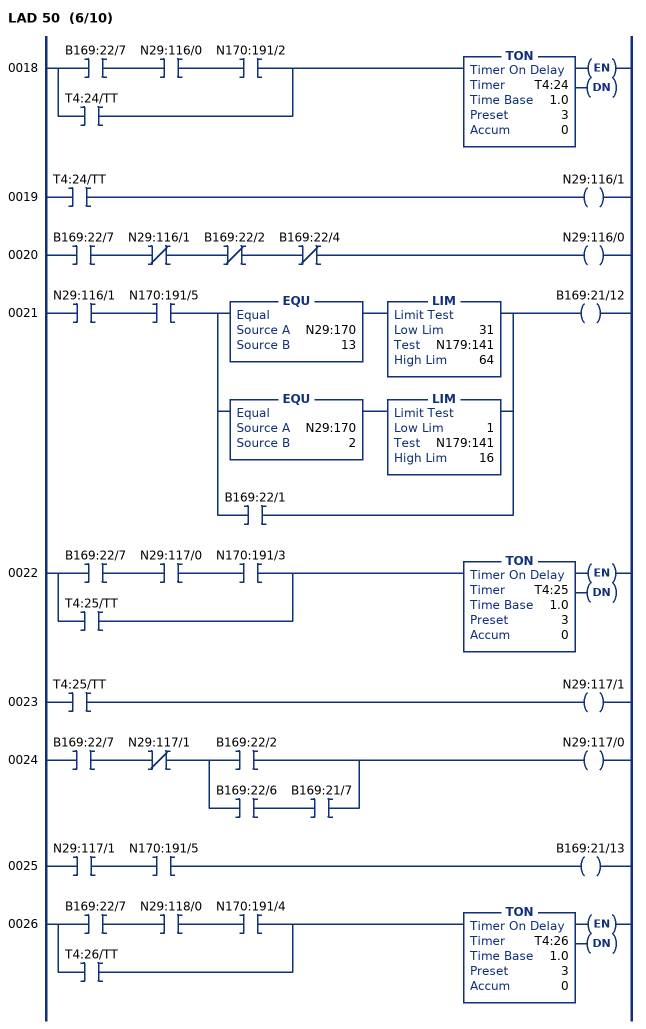
% Rung: 18 %
SOR BST XIC B169:22/7 XIC N29:116/0 XIC N170:191/2 NXB XIC T4:24/TT BND TON T4:24 1.0 3 0 EOR
% Rung: 19 %
SOR XIC T4:24/TT OTE N29:116/1 EOR
% Rung: 20 %
SOR XIC B169:22/7 XIO N29:116/1 XIO B169:22/2 XIO B169:22/4 OTE N29:116/0 EOR
% Rung: 21 %
SOR XIC N29:116/1 XIC N170:191/5 BST EQU N29:170 13 LIM 31 N179:141 64 NXB EQU N29:170 2 LIM 1 N179:141 16 NXB XIC B169:22/1 BND OTE B169:21/12 EOR
% Rung: 22 %
SOR BST XIC B169:22/7 XIC N29:117/0 XIC N170:191/3 NXB XIC T4:25/TT BND TON T4:25 1.0 3 0 EOR
% Rung: 23 %
SOR XIC T4:25/TT OTE N29:117/1 EOR
% Rung: 24 %
SOR XIC B169:22/7 XIO N29:117/1 BST XIC B169:22/2 NXB XIC B169:22/6 XIC B169:21/7 BND OTE N29:117/0 EOR
% Rung: 25 %
SOR XIC N29:117/1 XIC N170:191/5 OTE B169:21/13 EOR
% Rung: 26 %
SOR BST XIC B169:22/7 XIC N29:118/0 XIC N170:191/4 NXB XIC T4:26/TT BND TON T4:26 1.0 3 0 EOR

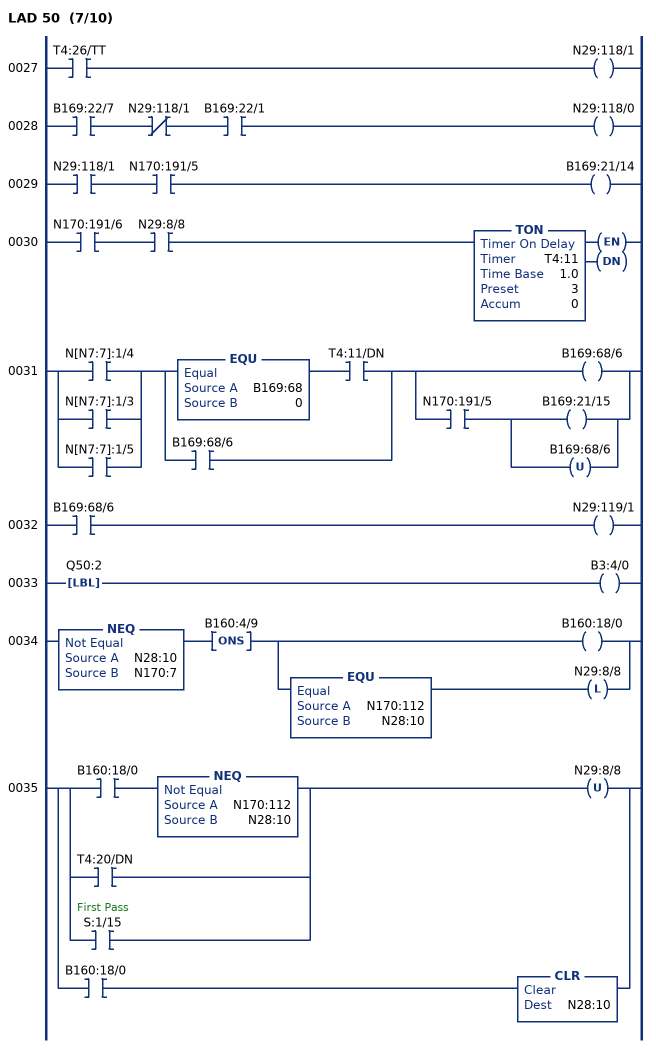
% Rung: 27 %
SOR XIC T4:26/TT OTE N29:118/1 EOR
% Rung: 28 %
SOR XIC B169:22/7 XIO N29:118/1 XIC B169:22/1 OTE N29:118/0 EOR
% Rung: 29 %
SOR XIC N29:118/1 XIC N170:191/5 OTE B169:21/14 EOR
% Rung: 30 %
SOR XIC N170:191/6 XIC N29:8/8 TON T4:11 1.0 3 0 EOR
% Rung: 31 %
SOR BST XIC N[N7:7]:1/4 NXB XIC N[N7:7]:1/3 NXB XIC N[N7:7]:1/5 BND BST EQU B169:68 0 XIC T4:11/DN NXB XIC B169:68/6 BND BST OTE B169:68/6 NXB XIC N170:191/5 BST OTE B169:21/15 NXB OTU B169:68/6 BND BND EOR
% Rung: 32 %
SOR XIC B169:68/6 OTE N29:119/1 EOR
% Rung: 33 %
SOR LBL Q50:2 OTE B3:4/0 EOR
% Rung: 34 %
SOR NEQ N28:10 N170:7 OSR B160:4/9 BST OTE B160:18/0 NXB EQU N170:112 N28:10 OTL N29:8/8 BND EOR
% Rung: 35 %
SOR BST BST XIC B160:18/0 NEQ N170:112 N28:10 NXB XIC T4:20/DN NXB XIC S:1/15 BND OTU N29:8/8 NXB XIC B160:18/0 CLR N28:10 BND EOR
%   S:1/15  "First Pass" %

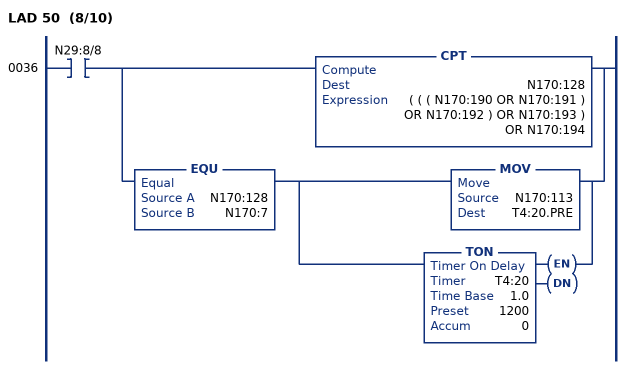
% Rung: 36 %
SOR XIC N29:8/8 BST CPT N170:128 " ( ( ( N170:190 OR N170:191 ) OR N170:192 ) OR N170:193 ) OR N170:194 " NXB EQU N170:128 N170:7 BST MOV N170:113 T4:20.PRE NXB TON T4:20 1.0 1200 0 BND BND EOR

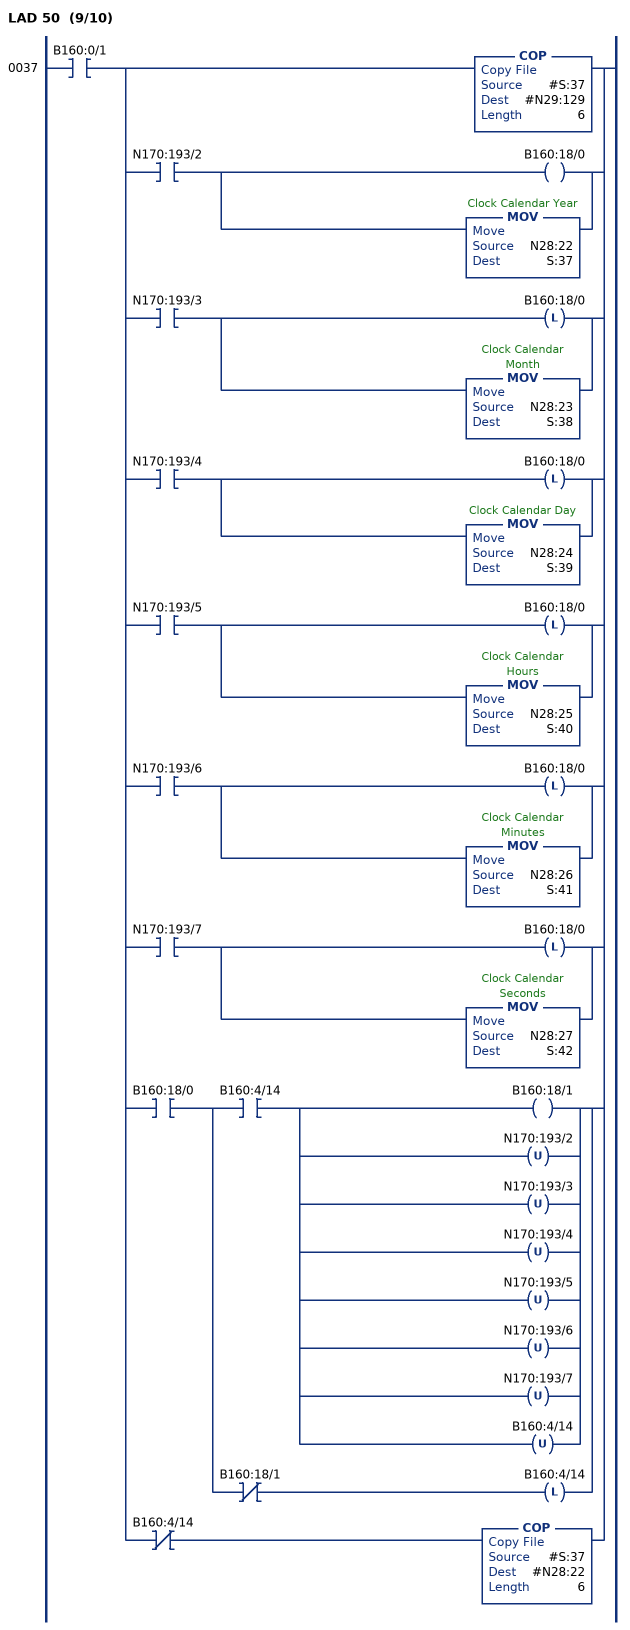
% Rung: 37 %
SOR XIC B160:0/1 BST COP #S:37 #N29:129 6 NXB XIC N170:193/2 BST OTE B160:18/0 NXB MOV N28:22 S:37 BND NXB XIC N170:193/3 BST OTL B160:18/0 NXB MOV N28:23 S:38 BND NXB XIC N170:193/4 BST OTL B160:18/0 NXB MOV N28:24 S:39 BND NXB XIC N170:193/5 BST OTL B160:18/0 NXB MOV N28:25 S:40 BND NXB XIC N170:193/6 BST OTL B160:18/0 NXB MOV N28:26 S:41 BND NXB XIC N170:193/7 BST OTL B160:18/0 NXB MOV N28:27 S:42 BND NXB XIC B160:18/0 BST XIC B160:4/14 BST OTE B160:18/1 NXB OTU N170:193/2 NXB OTU N170:193/3 NXB OTU N170:193/4 NXB OTU N170:193/5 NXB OTU N170:193/6 NXB OTU N170:193/7 NXB OTU B160:4/14 BND NXB XIO B160:18/1 OTL B160:4/14 BND NXB XIO B160:4/14 COP #S:37 #N28:22 6 BND EOR
%   S:37  "Clock Calendar Year" %
%   S:38  "Clock Calendar Month" %
%   S:39  "Clock Calendar Day" %
%   S:40  "Clock Calendar Hours" %
%   S:41  "Clock Calendar Minutes" %
%   S:42  "Clock Calendar Seconds" %

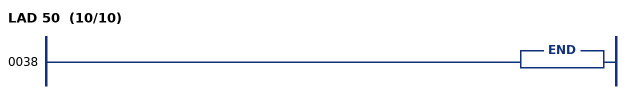
% Rung: 38 %
SOR END EOR

LADDER 51
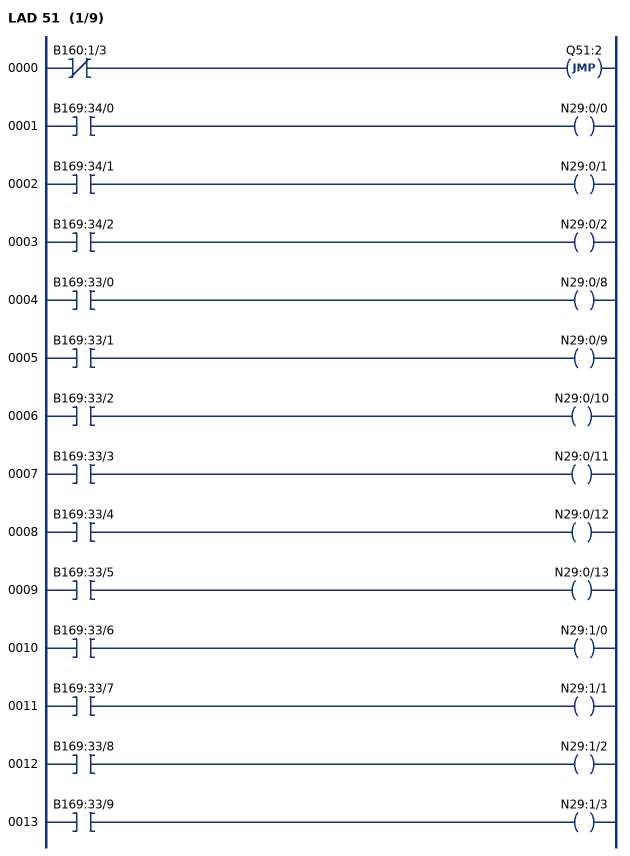
% Rung: 0 %
SOR XIO B160:1/3 JMP Q51:2 EOR
% Rung: 1 %
SOR XIC B169:34/0 OTE N29:0/0 EOR
% Rung: 2 %
SOR XIC B169:34/1 OTE N29:0/1 EOR
% Rung: 3 %
SOR XIC B169:34/2 OTE N29:0/2 EOR
% Rung: 4 %
SOR XIC B169:33/0 OTE N29:0/8 EOR
% Rung: 5 %
SOR XIC B169:33/1 OTE N29:0/9 EOR
% Rung: 6 %
SOR XIC B169:33/2 OTE N29:0/10 EOR
% Rung: 7 %
SOR XIC B169:33/3 OTE N29:0/11 EOR
% Rung: 8 %
SOR XIC B169:33/4 OTE N29:0/12 EOR
% Rung: 9 %
SOR XIC B169:33/5 OTE N29:0/13 EOR
% Rung: 10 %
SOR XIC B169:33/6 OTE N29:1/0 EOR
% Rung: 11 %
SOR XIC B169:33/7 OTE N29:1/1 EOR
% Rung: 12 %
SOR XIC B169:33/8 OTE N29:1/2 EOR
% Rung: 13 %
SOR XIC B169:33/9 OTE N29:1/3 EOR

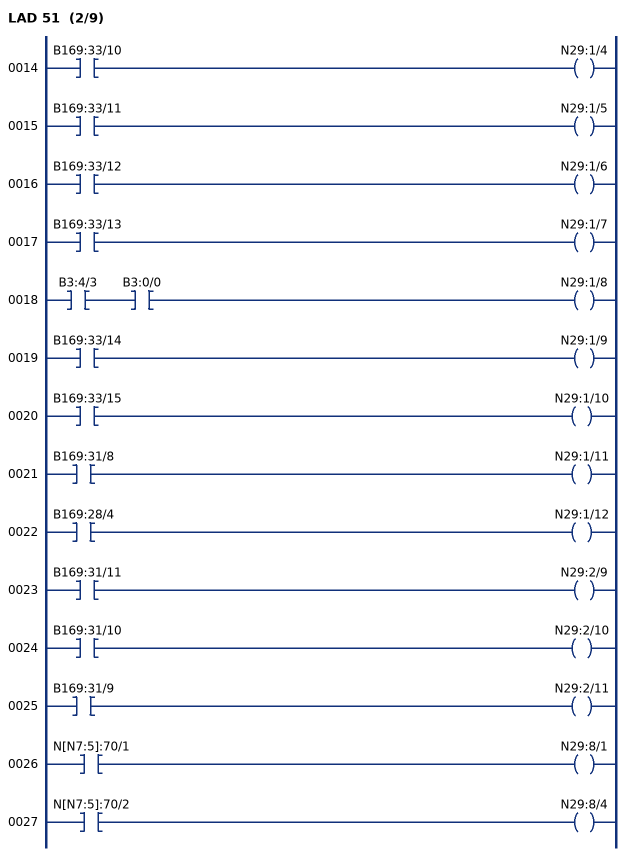
% Rung: 14 %
SOR XIC B169:33/10 OTE N29:1/4 EOR
% Rung: 15 %
SOR XIC B169:33/11 OTE N29:1/5 EOR
% Rung: 16 %
SOR XIC B169:33/12 OTE N29:1/6 EOR
% Rung: 17 %
SOR XIC B169:33/13 OTE N29:1/7 EOR
% Rung: 18 %
SOR XIC B3:4/3 XIC B3:0/0 OTE N29:1/8 EOR
% Rung: 19 %
SOR XIC B169:33/14 OTE N29:1/9 EOR
% Rung: 20 %
SOR XIC B169:33/15 OTE N29:1/10 EOR
% Rung: 21 %
SOR XIC B169:31/8 OTE N29:1/11 EOR
% Rung: 22 %
SOR XIC B169:28/4 OTE N29:1/12 EOR
% Rung: 23 %
SOR XIC B169:31/11 OTE N29:2/9 EOR
% Rung: 24 %
SOR XIC B169:31/10 OTE N29:2/10 EOR
% Rung: 25 %
SOR XIC B169:31/9 OTE N29:2/11 EOR
% Rung: 26 %
SOR XIC N[N7:5]:70/1 OTE N29:8/1 EOR
% Rung: 27 %
SOR XIC N[N7:5]:70/2 OTE N29:8/4 EOR

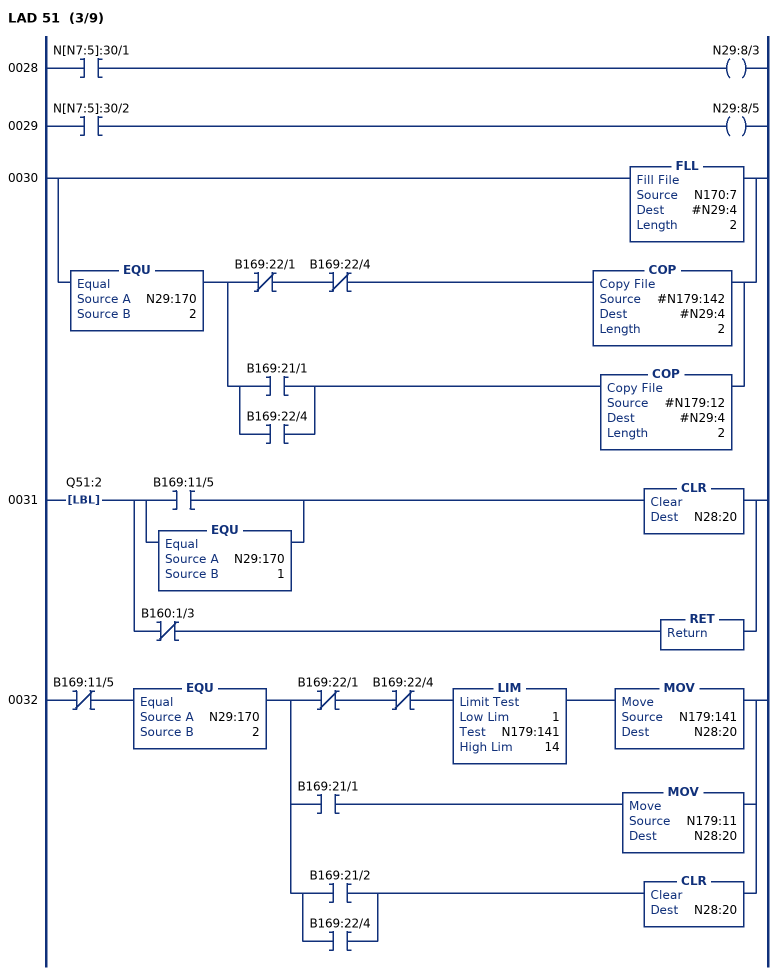
% Rung: 28 %
SOR XIC N[N7:5]:30/1 OTE N29:8/3 EOR
% Rung: 29 %
SOR XIC N[N7:5]:30/2 OTE N29:8/5 EOR
% Rung: 30 %
SOR BST FLL N170:7 #N29:4 2 NXB EQU N29:170 2 BST XIO B169:22/1 XIO B169:22/4 COP #N179:142 #N29:4 2 NXB BST XIC B169:21/1 NXB XIC B169:22/4 BND COP #N179:12 #N29:4 2 BND BND EOR
% Rung: 31 %
SOR LBL Q51:2 BST BST XIC B169:11/5 NXB EQU N29:170 1 BND CLR N28:20 NXB XIO B160:1/3 RET BND EOR
% Rung: 32 %
SOR XIO B169:11/5 EQU N29:170 2 BST XIO B169:22/1 XIO B169:22/4 LIM 1 N179:141 14 MOV N179:141 N28:20 NXB XIC B169:21/1 MOV N179:11 N28:20 NXB BST XIC B169:21/2 NXB XIC B169:22/4 BND CLR N28:20 BND EOR

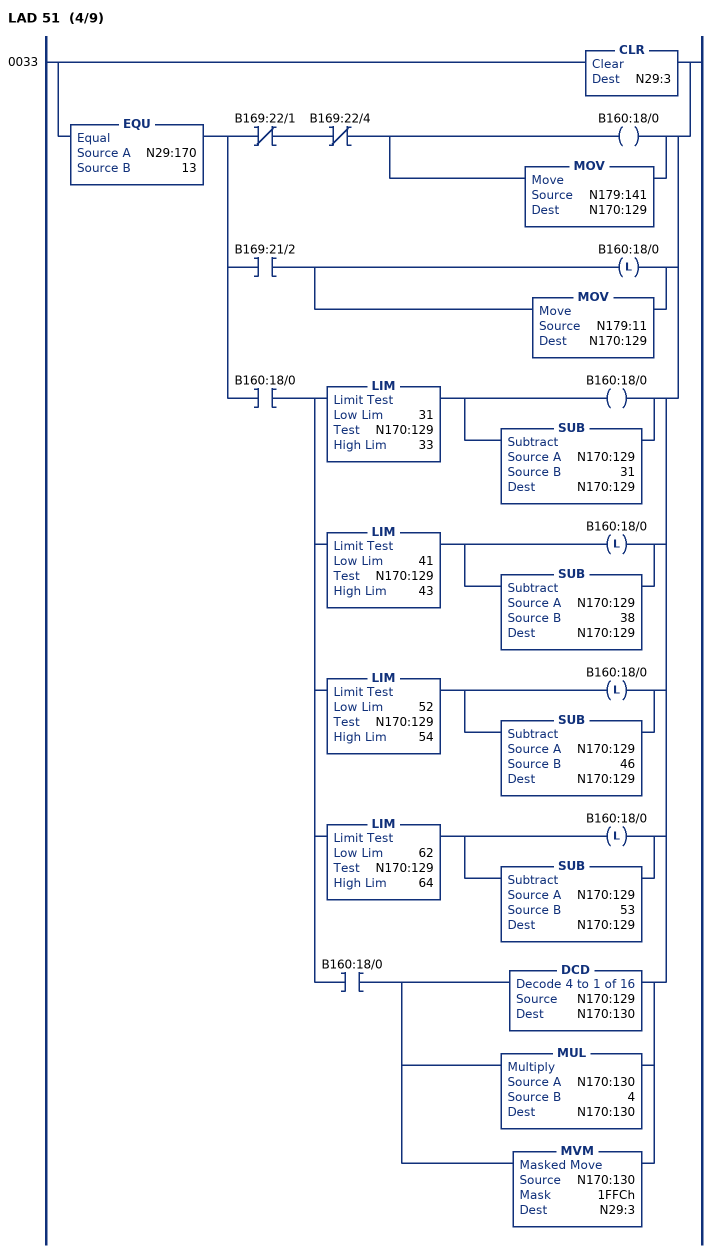
% Rung: 33 %
SOR BST CLR N29:3 NXB EQU N29:170 13 BST XIO B169:22/1 XIO B169:22/4 BST OTE B160:18/0 NXB MOV N179:141 N170:129 BND NXB XIC B169:21/2 BST OTL B160:18/0 NXB MOV N179:11 N170:129 BND NXB XIC B160:18/0 BST LIM 31 N170:129 33 BST OTE B160:18/0 NXB SUB N170:129 31 N170:129 BND NXB LIM 41 N170:129 43 BST OTL B160:18/0 NXB SUB N170:129 38 N170:129 BND NXB LIM 52 N170:129 54 BST OTL B160:18/0 NXB SUB N170:129 46 N170:129 BND NXB LIM 62 N170:129 64 BST OTL B160:18/0 NXB SUB N170:129 53 N170:129 BND NXB XIC B160:18/0 BST DCD N170:129 N170:130 NXB MUL N170:130 4 N170:130 NXB MVM N170:130 1FFCh N29:3 BND BND BND BND EOR

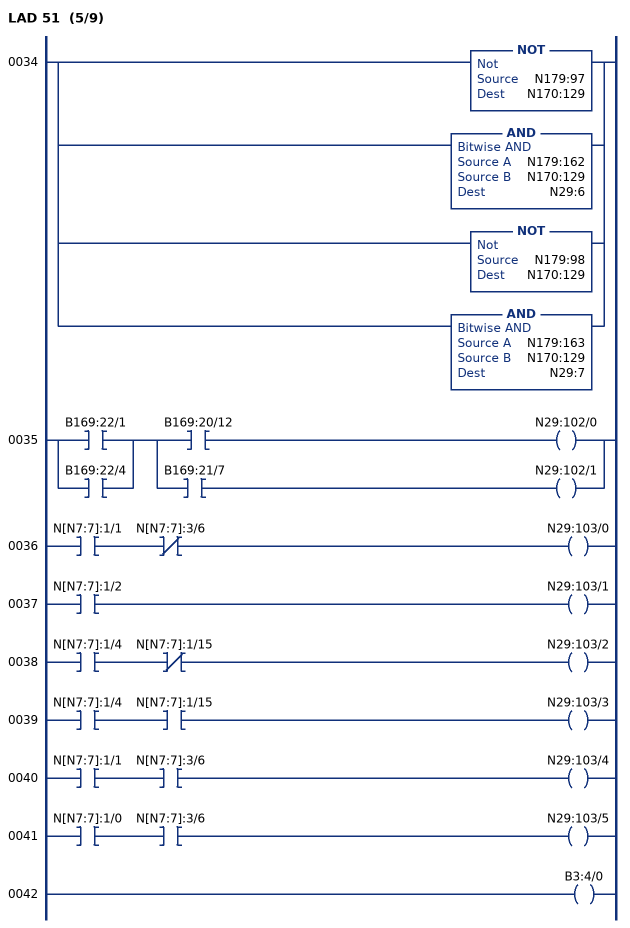
% Rung: 34 %
SOR BST NOT N179:97 N170:129 NXB AND N179:162 N170:129 N29:6 NXB NOT N179:98 N170:129 NXB AND N179:163 N170:129 N29:7 BND EOR
% Rung: 35 %
SOR BST XIC B169:22/1 NXB XIC B169:22/4 BND BST XIC B169:20/12 OTE N29:102/0 NXB XIC B169:21/7 OTE N29:102/1 BND EOR
% Rung: 36 %
SOR XIC N[N7:7]:1/1 XIO N[N7:7]:3/6 OTE N29:103/0 EOR
% Rung: 37 %
SOR XIC N[N7:7]:1/2 OTE N29:103/1 EOR
% Rung: 38 %
SOR XIC N[N7:7]:1/4 XIO N[N7:7]:1/15 OTE N29:103/2 EOR
% Rung: 39 %
SOR XIC N[N7:7]:1/4 XIC N[N7:7]:1/15 OTE N29:103/3 EOR
% Rung: 40 %
SOR XIC N[N7:7]:1/1 XIC N[N7:7]:3/6 OTE N29:103/4 EOR
% Rung: 41 %
SOR XIC N[N7:7]:1/0 XIC N[N7:7]:3/6 OTE N29:103/5 EOR
% Rung: 42 %
SOR OTE B3:4/0 EOR

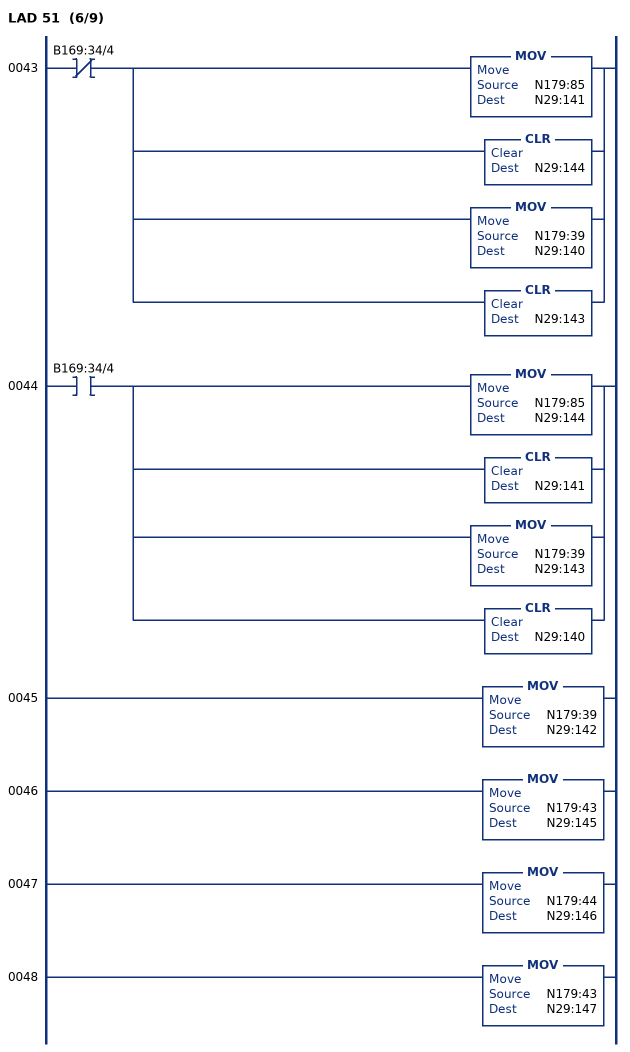
% Rung: 43 %
SOR XIO B169:34/4 BST MOV N179:85 N29:141 NXB CLR N29:144 NXB MOV N179:39 N29:140 NXB CLR N29:143 BND EOR
% Rung: 44 %
SOR XIC B169:34/4 BST MOV N179:85 N29:144 NXB CLR N29:141 NXB MOV N179:39 N29:143 NXB CLR N29:140 BND EOR
% Rung: 45 %
SOR MOV N179:39 N29:142 EOR
% Rung: 46 %
SOR MOV N179:43 N29:145 EOR
% Rung: 47 %
SOR MOV N179:44 N29:146 EOR
% Rung: 48 %
SOR MOV N179:43 N29:147 EOR

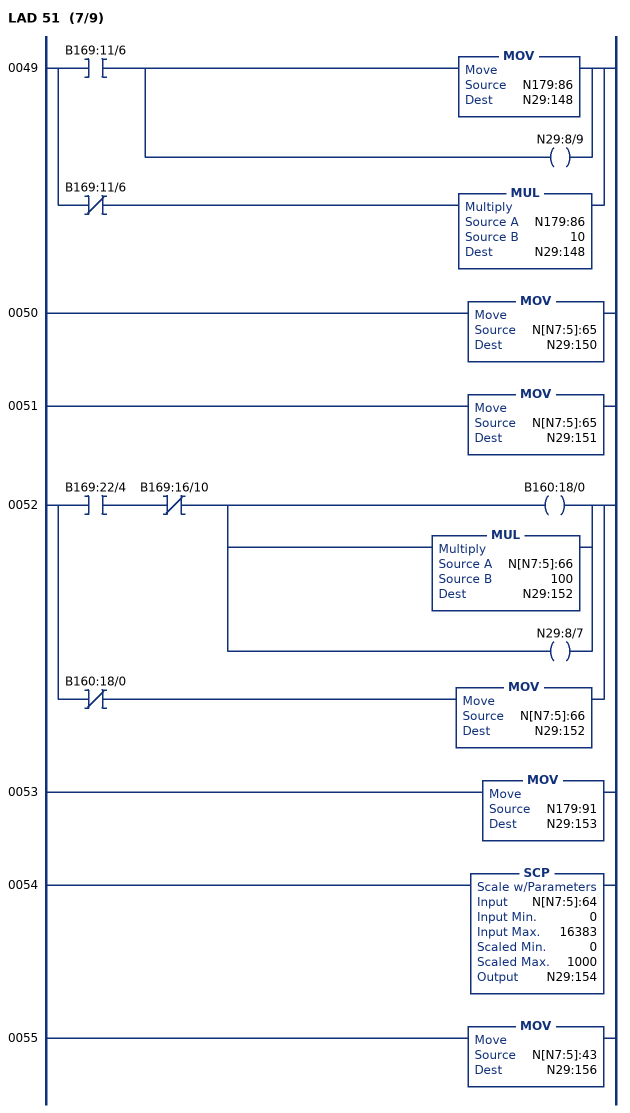
% Rung: 49 %
SOR BST XIC B169:11/6 BST MOV N179:86 N29:148 NXB OTE N29:8/9 BND NXB XIO B169:11/6 MUL N179:86 10 N29:148 BND EOR
% Rung: 50 %
SOR MOV N[N7:5]:65 N29:150 EOR
% Rung: 51 %
SOR MOV N[N7:5]:65 N29:151 EOR
% Rung: 52 %
SOR BST XIC B169:22/4 XIO B169:16/10 BST OTE B160:18/0 NXB MUL N[N7:5]:66 100 N29:152 NXB OTE N29:8/7 BND NXB XIO B160:18/0 MOV N[N7:5]:66 N29:152 BND EOR
% Rung: 53 %
SOR MOV N179:91 N29:153 EOR
% Rung: 54 %
SOR SCP N[N7:5]:64 0 16383 0 1000 N29:154 EOR
% Rung: 55 %
SOR MOV N[N7:5]:43 N29:156 EOR

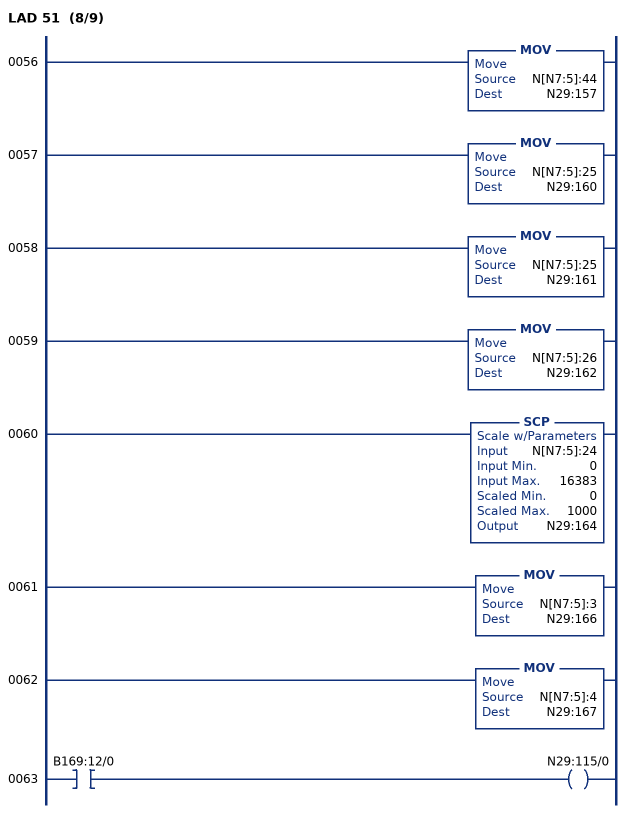
% Rung: 56 %
SOR MOV N[N7:5]:44 N29:157 EOR
% Rung: 57 %
SOR MOV N[N7:5]:25 N29:160 EOR
% Rung: 58 %
SOR MOV N[N7:5]:25 N29:161 EOR
% Rung: 59 %
SOR MOV N[N7:5]:26 N29:162 EOR
% Rung: 60 %
SOR SCP N[N7:5]:24 0 16383 0 1000 N29:164 EOR
% Rung: 61 %
SOR MOV N[N7:5]:3 N29:166 EOR
% Rung: 62 %
SOR MOV N[N7:5]:4 N29:167 EOR
% Rung: 63 %
SOR XIC B169:12/0 OTE N29:115/0 EOR

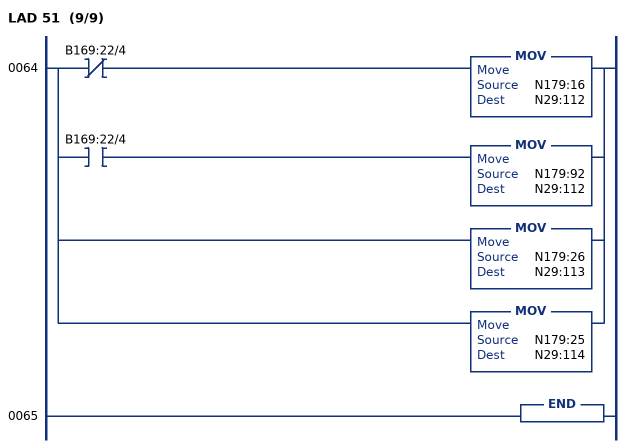
% Rung: 64 %
SOR BST BST XIO B169:22/4 MOV N179:16 N29:112 NXB XIC B169:22/4 MOV N179:92 N29:112 BND NXB MOV N179:26 N29:113 NXB MOV N179:25 N29:114 BND EOR
% Rung: 65 %
SOR END EOR

LADDER 52
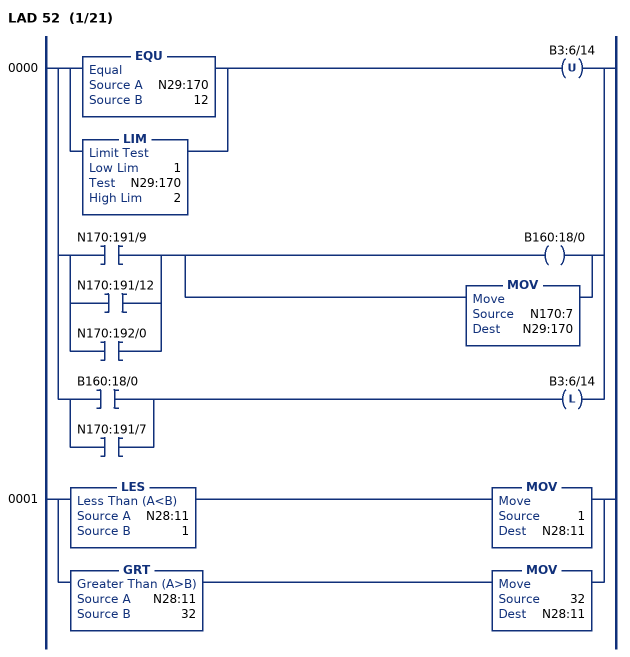
% Rung: 0 %
SOR BST BST EQU N29:170 12 NXB LIM 1 N29:170 2 BND OTU B3:6/14 NXB BST XIC N170:191/9 NXB XIC N170:191/12 NXB XIC N170:192/0 BND BST OTE B160:18/0 NXB MOV N170:7 N29:170 BND NXB BST XIC B160:18/0 NXB XIC N170:191/7 BND OTL B3:6/14 BND EOR
% Rung: 1 %
SOR BST LES N28:11 1 MOV 1 N28:11 NXB GRT N28:11 32 MOV 32 N28:11 BND EOR

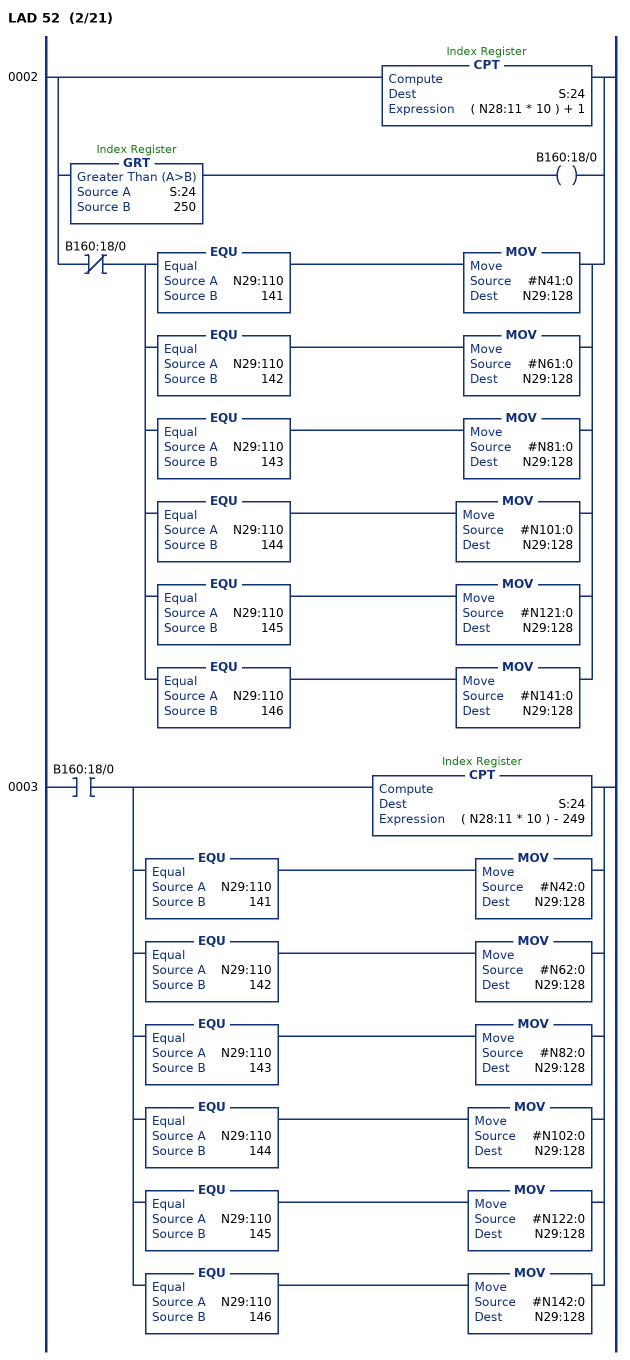
% Rung: 2 %
SOR BST CPT S:24 " ( N28:11 * 10 ) + 1 " NXB BST GRT S:24 250 OTE B160:18/0 NXB XIO B160:18/0 BST EQU N29:110 141 MOV #N41:0 N29:128 NXB EQU N29:110 142 MOV #N61:0 N29:128 NXB EQU N29:110 143 MOV #N81:0 N29:128 NXB EQU N29:110 144 MOV #N101:0 N29:128 NXB EQU N29:110 145 MOV #N121:0 N29:128 NXB EQU N29:110 146 MOV #N141:0 N29:128 BND BND BND EOR
%   S:24  "Index Register" %
% Rung: 3 %
SOR XIC B160:18/0 BST CPT S:24 " ( N28:11 * 10 ) - 249 " NXB EQU N29:110 141 MOV #N42:0 N29:128 NXB EQU N29:110 142 MOV #N62:0 N29:128 NXB EQU N29:110 143 MOV #N82:0 N29:128 NXB EQU N29:110 144 MOV #N102:0 N29:128 NXB EQU N29:110 145 MOV #N122:0 N29:128 NXB EQU N29:110 146 MOV #N142:0 N29:128 BND EOR
%   S:24  "Index Register" %

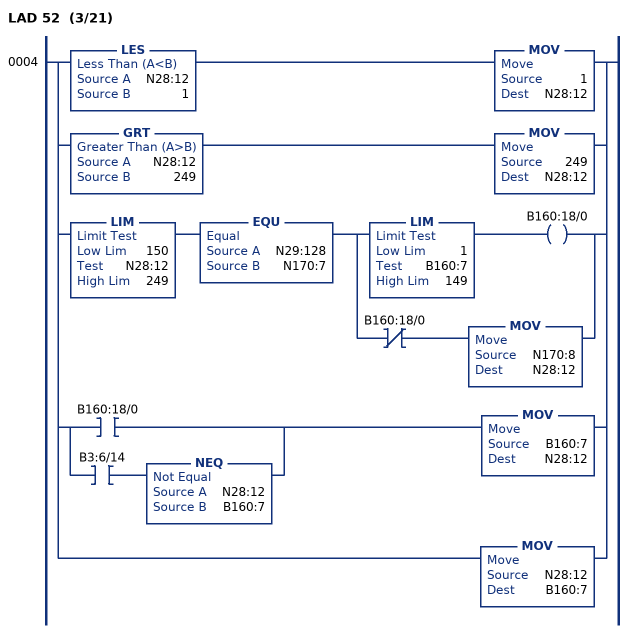
% Rung: 4 %
SOR BST LES N28:12 1 MOV 1 N28:12 NXB GRT N28:12 249 MOV 249 N28:12 NXB LIM 150 N28:12 249 EQU N29:128 N170:7 BST LIM 1 B160:7 149 OTE B160:18/0 NXB XIO B160:18/0 MOV N170:8 N28:12 BND NXB BST XIC B160:18/0 NXB XIC B3:6/14 NEQ N28:12 B160:7 BND MOV B160:7 N28:12 NXB MOV N28:12 B160:7 BND EOR

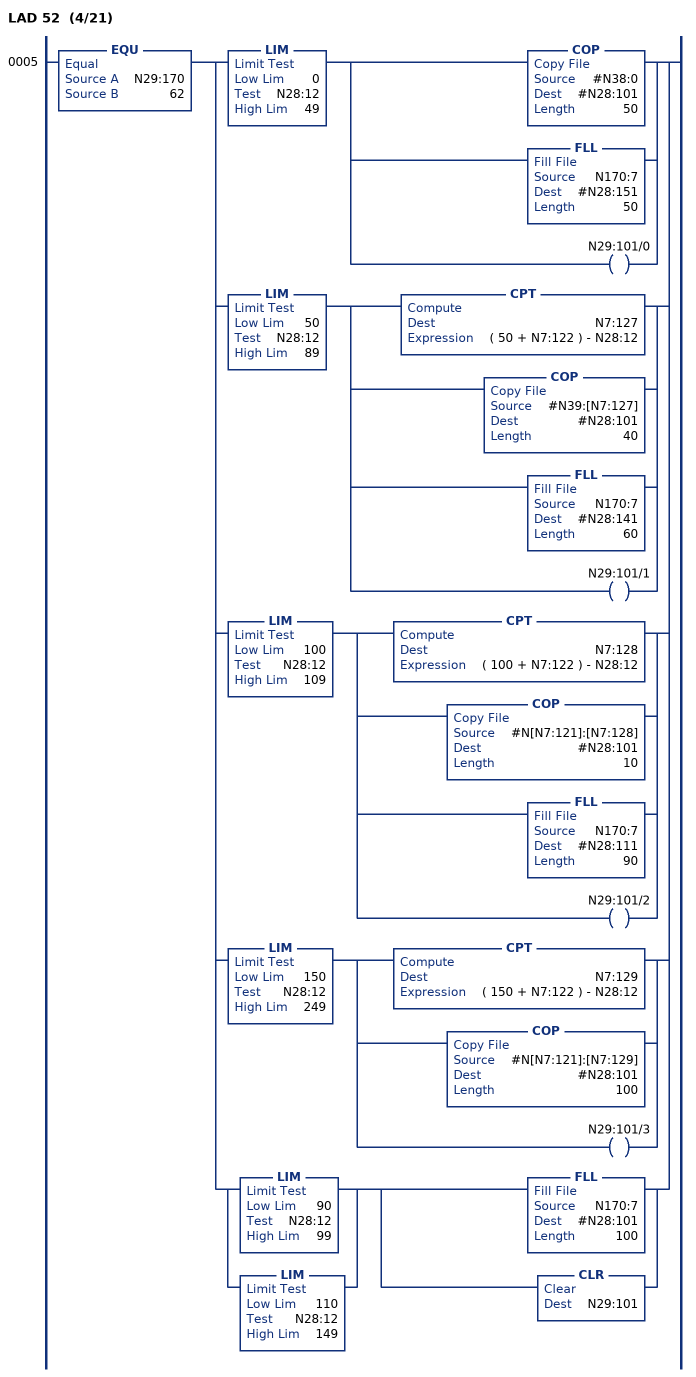
% Rung: 5 %
SOR EQU N29:170 62 BST LIM 0 N28:12 49 BST COP #N38:0 #N28:101 50 NXB FLL N170:7 #N28:151 50 NXB OTE N29:101/0 BND NXB LIM 50 N28:12 89 BST CPT N7:127 " ( 50 + N7:122 ) - N28:12 " NXB COP #N39:[N7:127] #N28:101 40 NXB FLL N170:7 #N28:141 60 NXB OTE N29:101/1 BND NXB LIM 100 N28:12 109 BST CPT N7:128 " ( 100 + N7:122 ) - N28:12 " NXB COP #N[N7:121]:[N7:128] #N28:101 10 NXB FLL N170:7 #N28:111 90 NXB OTE N29:101/2 BND NXB LIM 150 N28:12 249 BST CPT N7:129 " ( 150 + N7:122 ) - N28:12 " NXB COP #N[N7:121]:[N7:129] #N28:101 100 NXB OTE N29:101/3 BND NXB BST LIM 90 N28:12 99 NXB LIM 110 N28:12 149 BND BST FLL N170:7 #N28:101 100 NXB CLR N29:101 BND BND EOR

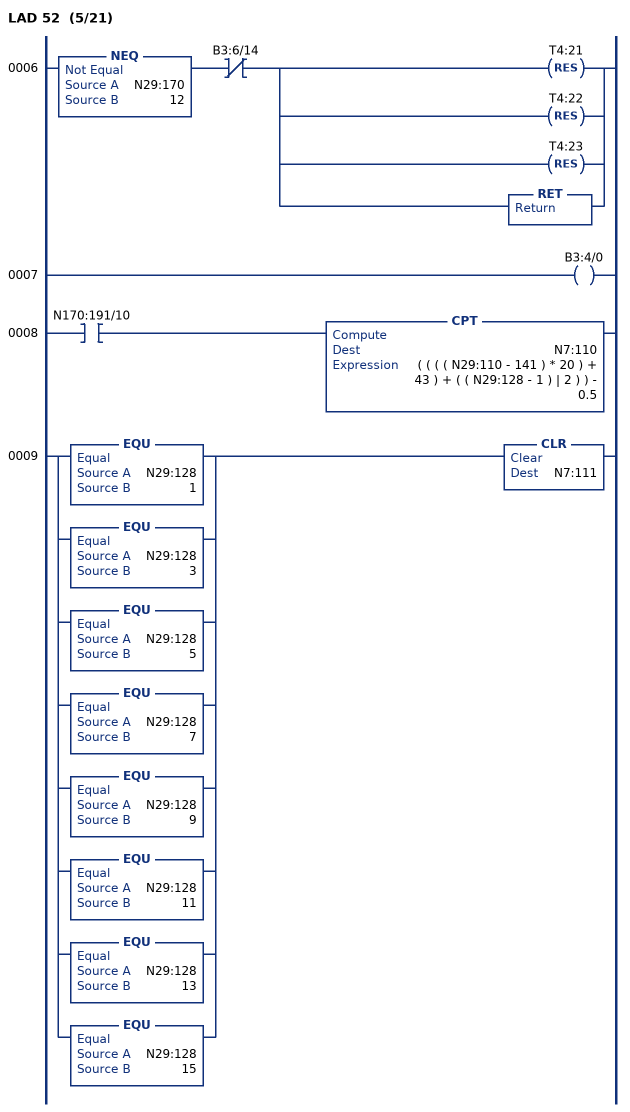
% Rung: 6 %
SOR NEQ N29:170 12 XIO B3:6/14 BST RES T4:21 NXB RES T4:22 NXB RES T4:23 NXB RET BND EOR
% Rung: 7 %
SOR OTE B3:4/0 EOR
% Rung: 8 %
SOR XIC N170:191/10 CPT N7:110 " ( ( ( ( N29:110 - 141 ) * 20 ) + 43 ) + ( ( N29:128 - 1 ) | 2 ) ) - 0.5 " EOR
% Rung: 9 %
SOR BST EQU N29:128 1 NXB EQU N29:128 3 NXB EQU N29:128 5 NXB EQU N29:128 7 NXB EQU N29:128 9 NXB EQU N29:128 11 NXB EQU N29:128 13 NXB EQU N29:128 15 BND CLR N7:111 EOR

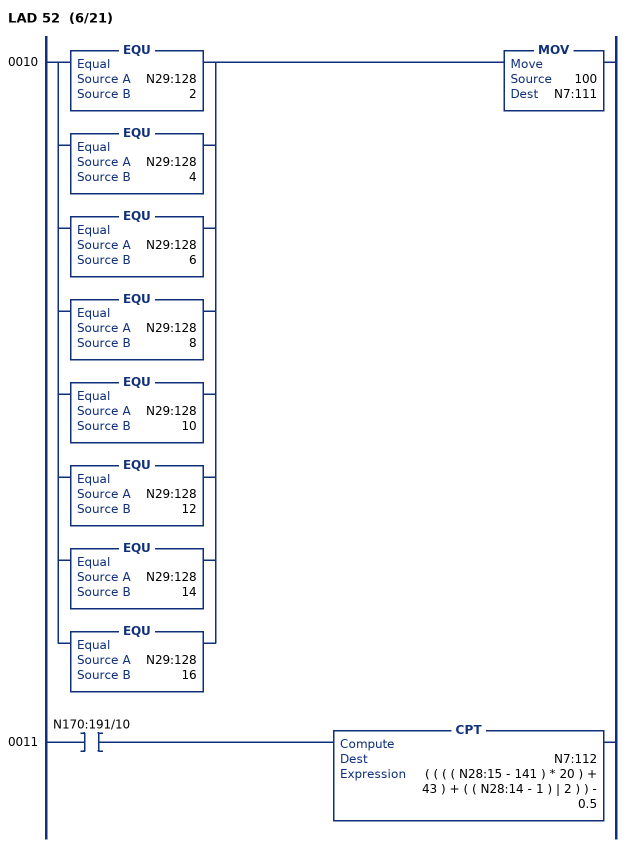
% Rung: 10 %
SOR BST EQU N29:128 2 NXB EQU N29:128 4 NXB EQU N29:128 6 NXB EQU N29:128 8 NXB EQU N29:128 10 NXB EQU N29:128 12 NXB EQU N29:128 14 NXB EQU N29:128 16 BND MOV 100 N7:111 EOR
% Rung: 11 %
SOR XIC N170:191/10 CPT N7:112 " ( ( ( ( N28:15 - 141 ) * 20 ) + 43 ) + ( ( N28:14 - 1 ) | 2 ) ) - 0.5 " EOR

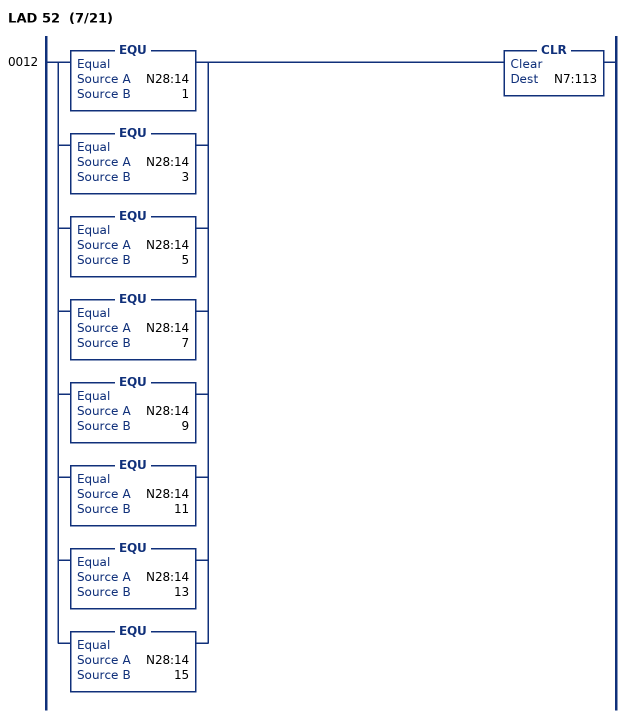
% Rung: 12 %
SOR BST EQU N28:14 1 NXB EQU N28:14 3 NXB EQU N28:14 5 NXB EQU N28:14 7 NXB EQU N28:14 9 NXB EQU N28:14 11 NXB EQU N28:14 13 NXB EQU N28:14 15 BND CLR N7:113 EOR

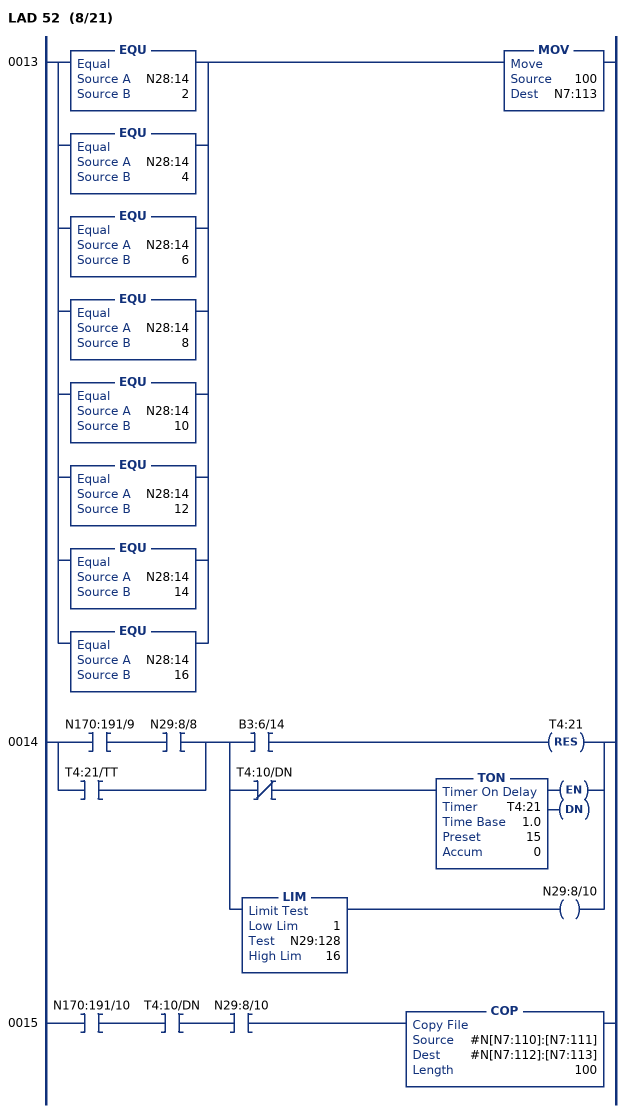
% Rung: 13 %
SOR BST EQU N28:14 2 NXB EQU N28:14 4 NXB EQU N28:14 6 NXB EQU N28:14 8 NXB EQU N28:14 10 NXB EQU N28:14 12 NXB EQU N28:14 14 NXB EQU N28:14 16 BND MOV 100 N7:113 EOR
% Rung: 14 %
SOR BST XIC N170:191/9 XIC N29:8/8 NXB XIC T4:21/TT BND BST XIC B3:6/14 RES T4:21 NXB XIO T4:10/DN TON T4:21 1.0 15 0 NXB LIM 1 N29:128 16 OTE N29:8/10 BND EOR
% Rung: 15 %
SOR XIC N170:191/10 XIC T4:10/DN XIC N29:8/10 COP #N[N7:110]:[N7:111] #N[N7:112]:[N7:113] 100 EOR

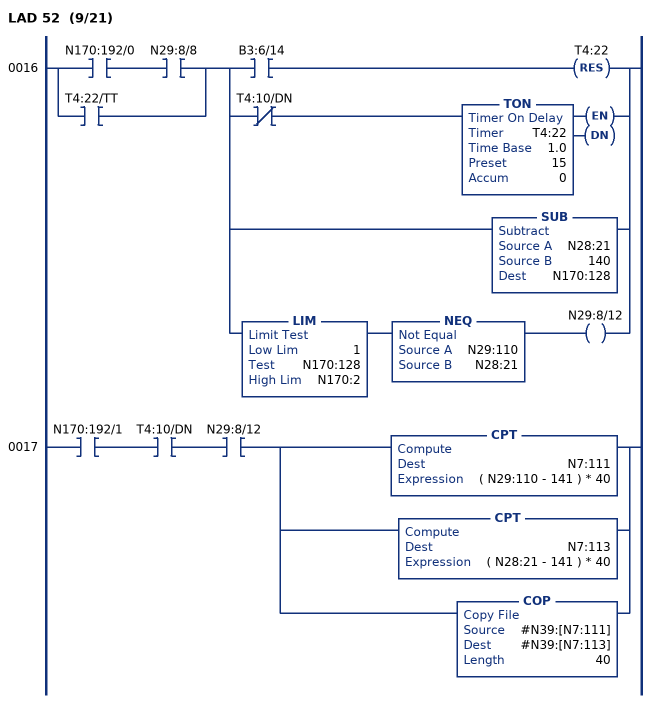
% Rung: 16 %
SOR BST XIC N170:192/0 XIC N29:8/8 NXB XIC T4:22/TT BND BST XIC B3:6/14 RES T4:22 NXB XIO T4:10/DN TON T4:22 1.0 15 0 NXB SUB N28:21 140 N170:128 NXB LIM 1 N170:128 N170:2 NEQ N29:110 N28:21 OTE N29:8/12 BND EOR
% Rung: 17 %
SOR XIC N170:192/1 XIC T4:10/DN XIC N29:8/12 BST CPT N7:111 " ( N29:110 - 141 ) * 40 " NXB CPT N7:113 " ( N28:21 - 141 ) * 40 " NXB COP #N39:[N7:111] #N39:[N7:113] 40 BND EOR

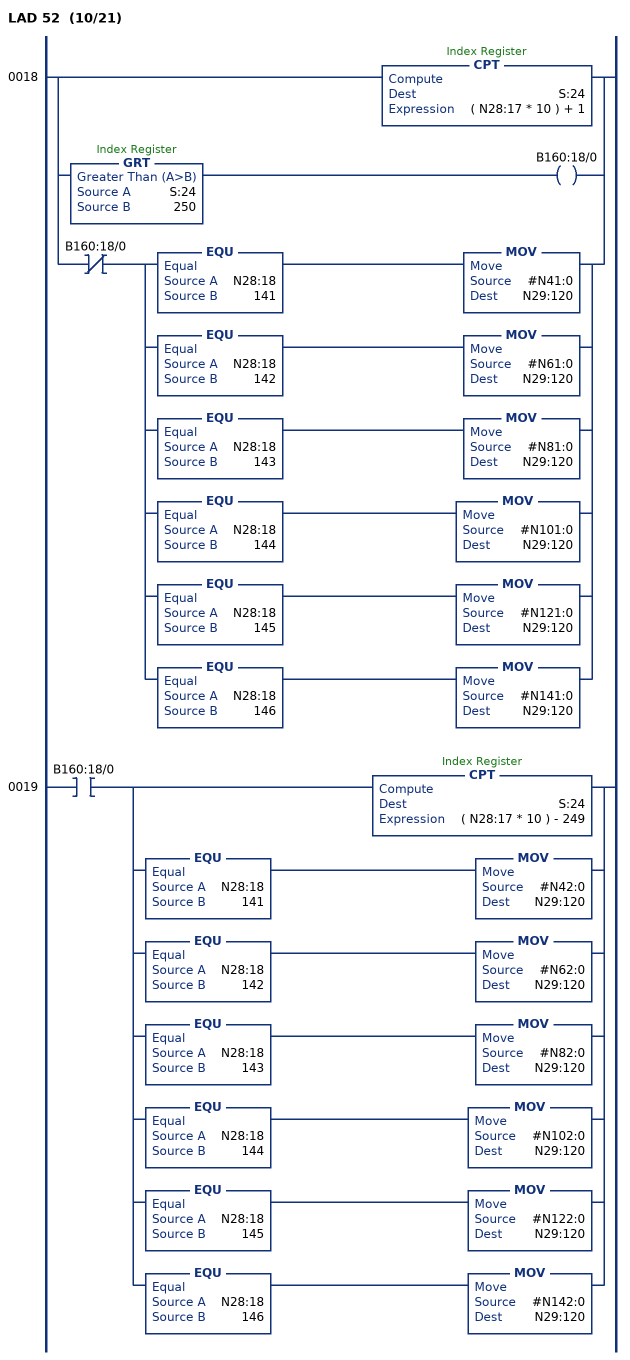
% Rung: 18 %
SOR BST CPT S:24 " ( N28:17 * 10 ) + 1 " NXB GRT S:24 250 OTE B160:18/0 NXB XIO B160:18/0 BST EQU N28:18 141 MOV #N41:0 N29:120 NXB EQU N28:18 142 MOV #N61:0 N29:120 NXB EQU N28:18 143 MOV #N81:0 N29:120 NXB EQU N28:18 144 MOV #N101:0 N29:120 NXB EQU N28:18 145 MOV #N121:0 N29:120 NXB EQU N28:18 146 MOV #N141:0 N29:120 BND BND EOR
%   S:24  "Index Register" %
% Rung: 19 %
SOR XIC B160:18/0 BST CPT S:24 " ( N28:17 * 10 ) - 249 " NXB EQU N28:18 141 MOV #N42:0 N29:120 NXB EQU N28:18 142 MOV #N62:0 N29:120 NXB EQU N28:18 143 MOV #N82:0 N29:120 NXB EQU N28:18 144 MOV #N102:0 N29:120 NXB EQU N28:18 145 MOV #N122:0 N29:120 NXB EQU N28:18 146 MOV #N142:0 N29:120 BND EOR
%   S:24  "Index Register" %

